FUNCTION_BLOCK FB_SetEnables
VAR_IN_OUT
	stMotionStage: DUT_MotionStage;
END_VAR

stMotionStage.bAllForwardEnable := stMotionStage.bLimitForwardEnable AND (stMotionStage.bGantryForwardEnable OR NOT stMotionStage.bGantryAxis);
stMotionStage.bAllBackwardEnable := stMotionStage.bLimitBackwardEnable AND (stMotionStage.bGantryBackwardEnable OR NOT stMotionStage.bGantryAxis);

stMotionStage.bAllEnable := stMotionStage.bEnable AND stMotionStage.bHardwareEnable;

END_FUNCTION_BLOCK

(* stored: Version 1.1.0.1, ProductVersion 3.1.4022.12
   POU FB_SetEnables: Id {9028a506-3476-4ab7-9f18-be1b77c07efa}, SpecialFunc None *)
